// LS Electric XG5000 project: p833
// PLC NewPLC
// module base 0 slot 0: 입출력 모듈:XBM-DN32H (DC 24V입력/TR 출력, 32점)

PROGRAM NewProgram (task: 스캔 프로그램)

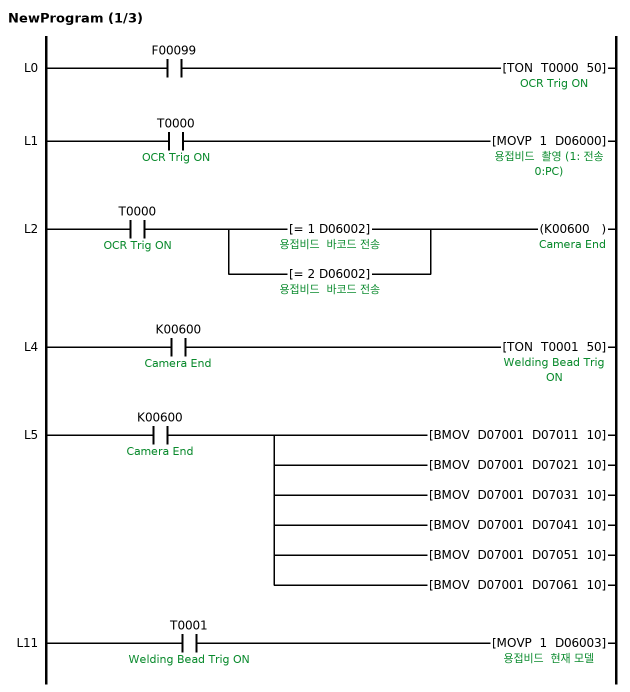
; L0
LOAD      F00099
TON       T0000 50	// OCR Trig ON
; L1
LOAD      T0000	// OCR Trig ON
MOVP      1 D06000	// 용접비드  촬영 (1: 전송 0:PC)
; L2
LOAD      T0000	// OCR Trig ON
LOAD=     1 D06002	// 용접비드  바코드 전송
OR=       2 D06002	// 용접비드  바코드 전송
AND LOAD
OUT       K00600	// Camera End
; L4
LOAD      K00600	// Camera End
TON       T0001 50	// Welding Bead Trig ON
; L5
LOAD      K00600	// Camera End
BMOV      D07001 D07011 10
BMOV      D07001 D07021 10
BMOV      D07001 D07031 10
BMOV      D07001 D07041 10
BMOV      D07001 D07051 10
BMOV      D07001 D07061 10
; L11
LOAD      T0001	// Welding Bead Trig ON
MOVP      1 D06003	// 용접비드  현재 모델

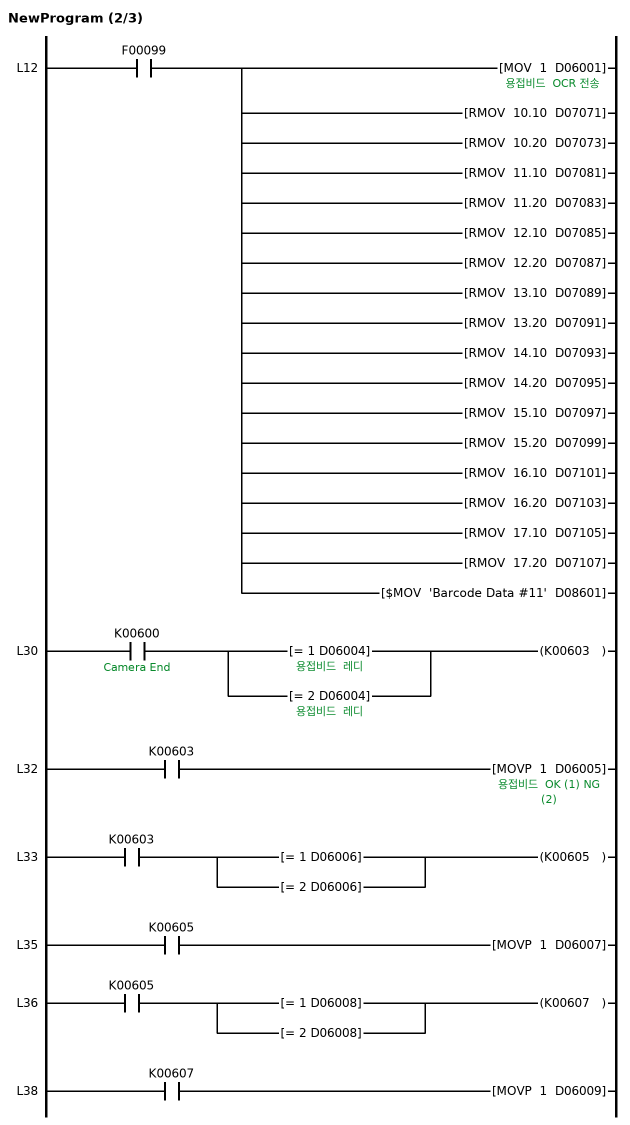
; L12
LOAD      F00099
MOV       1 D06001	// 용접비드  OCR 전송
RMOV      10.10 D07071
RMOV      10.20 D07073
RMOV      11.10 D07081
RMOV      11.20 D07083
RMOV      12.10 D07085
RMOV      12.20 D07087
RMOV      13.10 D07089
RMOV      13.20 D07091
RMOV      14.10 D07093
RMOV      14.20 D07095
RMOV      15.10 D07097
RMOV      15.20 D07099
RMOV      16.10 D07101
RMOV      16.20 D07103
RMOV      17.10 D07105
RMOV      17.20 D07107
$MOV      'Barcode Data #11' D08601
; L30
LOAD      K00600	// Camera End
LOAD=     1 D06004	// 용접비드  레디 
OR=       2 D06004	// 용접비드  레디 
AND LOAD
OUT       K00603
; L32
LOAD      K00603
MOVP      1 D06005	// 용접비드  OK (1) NG (2)
; L33
LOAD      K00603
LOAD=     1 D06006
OR=       2 D06006
AND LOAD
OUT       K00605
; L35
LOAD      K00605
MOVP      1 D06007
; L36
LOAD      K00605
LOAD=     1 D06008
OR=       2 D06008
AND LOAD
OUT       K00607
; L38
LOAD      K00607
MOVP      1 D06009

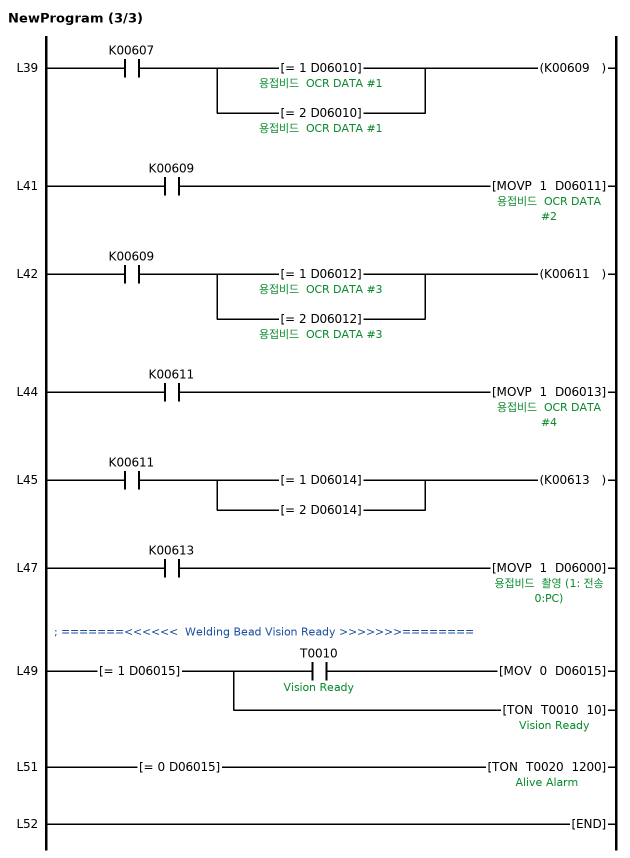
; L39
LOAD      K00607
LOAD=     1 D06010	// 용접비드  OCR DATA #1
OR=       2 D06010	// 용접비드  OCR DATA #1
AND LOAD
OUT       K00609
; L41
LOAD      K00609
MOVP      1 D06011	// 용접비드  OCR DATA #2
; L42
LOAD      K00609
LOAD=     1 D06012	// 용접비드  OCR DATA #3
OR=       2 D06012	// 용접비드  OCR DATA #3
AND LOAD
OUT       K00611
; L44
LOAD      K00611
MOVP      1 D06013	// 용접비드  OCR DATA #4
; L45
LOAD      K00611
LOAD=     1 D06014
OR=       2 D06014
AND LOAD
OUT       K00613
; L47
LOAD      K00613
MOVP      1 D06000	// 용접비드  촬영 (1: 전송 0:PC)
// =======<<<<<<  Welding Bead Vision Ready >>>>>>>========
; L49
LOAD=     1 D06015
MPUSH
AND       T0010	// Vision Ready
MOV       0 D06015
MPOP
TON       T0010 10	// Vision Ready
; L51
LOAD=     0 D06015
TON       T0020 1200	// Alive Alarm
; L52
END

VARIABLES AND COMMENTS (devices not used above)
K00591	BIT	CAR TYPE TMA 2WD
K00592	BIT	CAR TYPE TMA 4WD
K00593	BIT	CAR TYPE ON 2WD
K00594	BIT	CAR TYPE ON 4WD
T0002	BIT/WORD	Trig OFF
P00020	BIT	OCR Trig
P00021	BIT	Visin Trig
D06020	WORD	용접비드  바코드 #1
D04010	WORD	용접 비드 OCR
D04020	WORD	용접 바코드